// TIA Portal V21 export
DATA_BLOCK "UnitTestsDB"   // DB1
// stored: InstanceOfName UnitTests, InstanceOfType FB
"UnitTests"
   // VAR
   //    motorSim { S7_SetPoint := 'True'} : "MotorSim";
   //    motor1 { S7_SetPoint := 'True'} : "MotorControl";
   //    motor1Interface { S7_SetPoint := 'True'} : "motorInterface";
   //    motor1Config { S7_SetPoint := 'True'} : "motorConfig";
   //    motor1Hmi { S7_SetPoint := 'True'} : "motorHMI";
   //    switchgearSim { S7_SetPoint := 'True'} : "SwitchgearSim";
   //    switchgear1 { S7_SetPoint := 'True'} : "SwitchgearControl";
   //    switchgear1Interface { S7_SetPoint := 'True'} : "switchgearInterface";
   //    switchgear1Cfg { S7_SetPoint := 'True'} : "switchgearConfig";
   //    switchgear1Hmi { S7_SetPoint := 'True'} : "switchgearHMI";
   //    twoStepController { S7_SetPoint := 'True'} : "TwoStepController";
   //    prevSysTime : Time;
   //    resTimer { S7_SetPoint := 'True'} : "ResTONdt";
   //    preStartAlarm { S7_SetPoint := 'True'} : "PreStartAlarm";
   //    FOTDTimer : Time;
   //    FOTDModel { S7_SetPoint := 'True'} : "Fotd";
   // END_VAR
BEGIN
END_DATA_BLOCK
